// TIA Portal V17 export
// export: Created 2023-12-22T15:04:41.0781362Z, ExportSetting WithDefaults, DisplayName Totally Integrated Automation Portal, DisplayVersion V17, DisplayName TIA Portal Openness, DisplayVersion V17, DisplayName TIA Portal Version Control Interface, DisplayVersion V17, DisplayName STEP 7 Professional, DisplayVersion V17, DisplayName STEP 7 Safety, DisplayVersion V17, DisplayName WinCC Advanced, DisplayVersion V17
FUNCTION_BLOCK "DIx_1"   // FB200, LAD
{ S7_Optimized_Access := 'FALSE' }
VERSION : 0.1
// Input - входной сигнал контроллера
// pulse - частота фильтрации дребезга
// Signal - обработанный и отфильтрованный сигнал, используемый в дальнейшем
// stored: AutoNumber false, IsIECCheckEnabled false, SetENOAutomatically false, UDAEnableTagReadback false
   VAR
      AllBlock { S7_SetPoint := 'True'} : "DI_ex";   // Аварийный останов / 2.4 разрешение на работу
      "3FOk" { S7_SetPoint := 'True'} : "DI_ex";   // Питание в норме / 2.3 Нижний уровень
      Pump_Alarm { S7_SetPoint := 'True'} : "DI_ex";   // Авария насоса / Ротаметр 1
      Leak_KP { S7_SetPoint := 'True'} : "DI_ex";   // Затопление камеры КП2.7 / Ротаметр 2
      Level_Norm { S7_SetPoint := 'True'} : "DI_ex";   // Уровень в норме / Ротаметр 3
      "3Fok_1" { S7_SetPoint := 'True'} : "DI_ex";   // 3ф. сети Ввод 1 в норме / Датчик переливва
      "3Fok_2" { S7_SetPoint := 'True'} : "DI_ex";   // 3ф. сети Ввод 2 в норме / Датчик переливва
      "3Fok_sh" { S7_SetPoint := 'True'} : "DI_ex";   // 3ф. сети Ввод Шин в норме
      SHUSKV_Ok { S7_SetPoint := 'True'} : "DI_ex";   // Выключатель UC. Питание ШУСКВ в норме
      Leak_KP_res { S7_SetPoint := 'True'} : "DI_ex";
      Leak_KP_res_1 { S7_SetPoint := 'True'} : "DI_ex";
      signal_12 { S7_SetPoint := 'True'} : "DI_ex";
   END_VAR
   VAR DB_SPECIFIC
      Time_DTL { S7_SetPoint := 'True'} : DTL;
   END_VAR
   // AllBlock.ADDR_Bit := 3;
   // "3FOk".ADDR_Bit := 0;
   // Pump_Alarm.ADDR_Bit := 2;
   // Leak_KP.ADDR_Bit := 4;
   // Level_Norm.ADDR_Bit := 5;
   // "3Fok_1".ADDR_Bit := 6;
   // "3Fok_2".ADDR_Bit := 7;
   // "3Fok_sh".ADDR_Byte := 1;
   // "3Fok_sh".ADDR_Bit := 0;
   // SHUSKV_Ok.ADDR_Byte := 1;
   // SHUSKV_Ok.ADDR_Bit := 1;
   // Leak_KP_res.ADDR_Byte := 1;
   // Leak_KP_res.ADDR_Bit := 2;
   // Leak_KP_res_1.ADDR_Byte := 1;
   // Leak_KP_res_1.ADDR_Bit := 3;
   VAR_TEMP   // added for the SCL form of the ladder/FBD networks
      _w1 : Bool;
   END_VAR
BEGIN

REGION Network 1: AllBlock
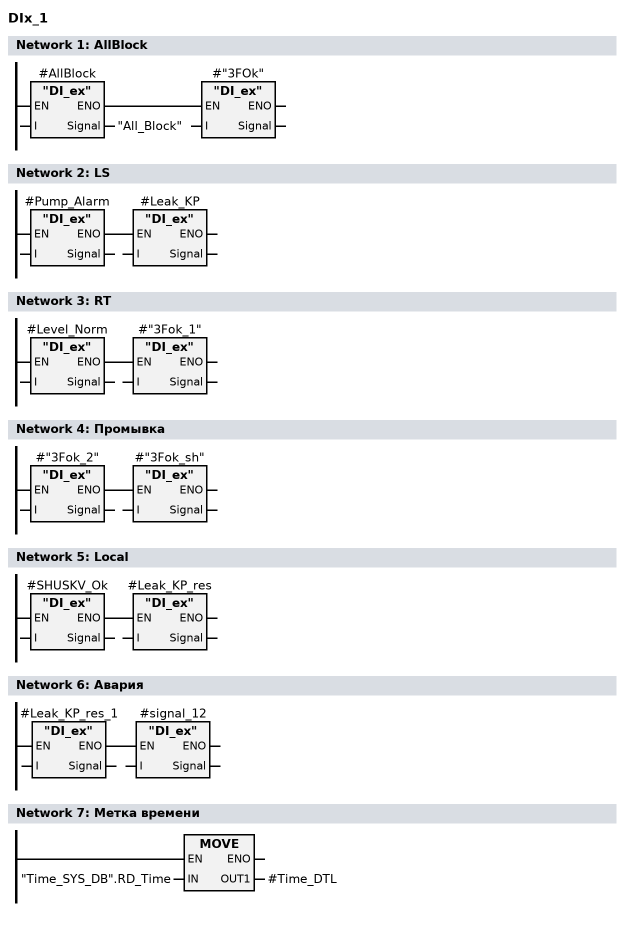
   RUNG wire#powerrail
      #AllBlock(I :=, Signal => "All_Block")
      #"3FOk"(I :=, Signal =>)
   END_RUNG
   // the same network as SCL:
   #AllBlock(Signal => "All_Block", ENO => #_w1);   // "DI_ex"
   IF #_w1 THEN
       #"3FOk"();   // "DI_ex"
   END_IF;
END_REGION

REGION Network 2: LS
   RUNG wire#powerrail
      #Pump_Alarm(I :=, Signal =>)
      #Leak_KP(I :=, Signal =>)
   END_RUNG
   // the same network as SCL:
   #Pump_Alarm(ENO => #_w1);   // "DI_ex"
   IF #_w1 THEN
       #Leak_KP();   // "DI_ex"
   END_IF;
END_REGION

REGION Network 3: RT
   RUNG wire#powerrail
      #Level_Norm(I :=, Signal =>)
      #"3Fok_1"(I :=, Signal =>)
   END_RUNG
   // the same network as SCL:
   #Level_Norm(ENO => #_w1);   // "DI_ex"
   IF #_w1 THEN
       #"3Fok_1"();   // "DI_ex"
   END_IF;
END_REGION

REGION Network 4: Промывка
   RUNG wire#powerrail
      #"3Fok_2"(I :=, Signal =>)
      #"3Fok_sh"(I :=, Signal =>)
   END_RUNG
   // the same network as SCL:
   #"3Fok_2"(ENO => #_w1);   // "DI_ex"
   IF #_w1 THEN
       #"3Fok_sh"();   // "DI_ex"
   END_IF;
END_REGION

REGION Network 5: Local
   RUNG wire#powerrail
      #SHUSKV_Ok(I :=, Signal =>)
      #Leak_KP_res(I :=, Signal =>)
   END_RUNG
   // the same network as SCL:
   #SHUSKV_Ok(ENO => #_w1);   // "DI_ex"
   IF #_w1 THEN
       #Leak_KP_res();   // "DI_ex"
   END_IF;
END_REGION

REGION Network 6: Авария
   RUNG wire#powerrail
      #Leak_KP_res_1(I :=, Signal =>)
      #signal_12(I :=, Signal =>)
   END_RUNG
   // the same network as SCL:
   #Leak_KP_res_1(ENO => #_w1);   // "DI_ex"
   IF #_w1 THEN
       #signal_12();   // "DI_ex"
   END_IF;
END_REGION

REGION Network 7: Метка времени
   RUNG wire#powerrail
      Move(in := "Time_SYS_DB".RD_Time, out1 => #Time_DTL)
   END_RUNG
   // the same network as SCL:
   #Time_DTL := "Time_SYS_DB".RD_Time;
END_REGION
END_FUNCTION_BLOCK
